KUKA KRL program: kvp_interface.src

&ACCESS RV
&PARAM TPVW_VERSION =3.3.5
&COMMENT KVP Interface
&REL 1
DEF kvp_interface( )
; This program is used to initialize the KVP interface and ensure that the system is ready for operation.
; It sets up the necessary parameters and waits for the system to be ready.
; Make sure the program is not called by a selection

;Make a notify message to be sure that the program is running

END
